TYPE IOExpantionMessageSubData_t :
STRUCT
	callbackVariable : POINTER TO BOOL := NULL;
	messageDescription : IOExpantionMessageDescriptor_t;
END_STRUCT
END_TYPE

(* stored: Version 1.1.0.1
   DUT IOExpantionMessageSubData_t: Id {0b4f4dfd-4df0-4db2-80cf-d6545774dc3c} *)
